TYPE U_Convert :  
	UNION  
		arrUDP_Data: ARRAY [0 .. 3] OF BYTE; // Array must start with LSB  
		rReal : REAL;  
	END_UNION  
END_TYPE

(* stored: Version 1.1.0.1, ProductVersion 3.1.4024.12
   POU U_Convert: Id {135bad39-a65a-4041-aed8-a9b22fd39e15}, SpecialFunc None *)
